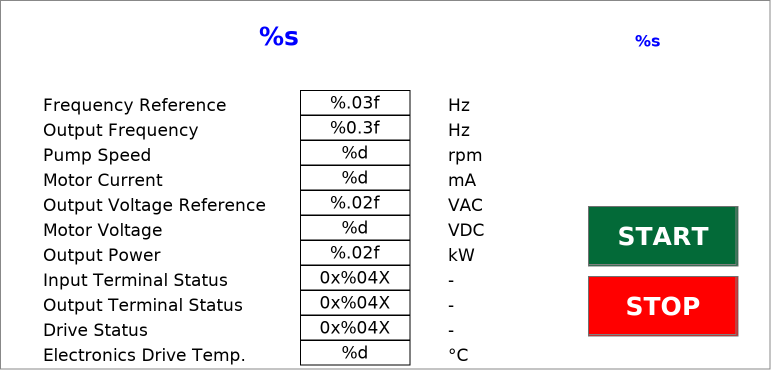
VISUALIZATION GUI_TEMPLATE_ECODRY_V01  // 771x370
VAR_IN_OUT
	m_Instance:	FB_CRYO_PUMP_ECODRY;
	m_bEnable:	BOOL;	// Flag to start/stop the pump
END_VAR
    Rectangle (300,90 110x25), "%.03f", text variable: m_Instance.stat.lrFreqRef
    Rectangle (300,115 110x25), "%0.3f", text variable: m_Instance.stat.lrOutFreq
    Rectangle (300,165 110x25), "%d", text variable: m_Instance.stat.nMotorCurr
    Rectangle (300,190 110x25), "%.02f", text variable: m_Instance.stat.lrOutVoltRef
    Label (40,90 245x30), "Frequency Reference"
    Label (40,115 245x30), "Output Frequency"
    Label (40,165 245x30), "Motor Current"
    Label (40,190 245x30), "Output Voltage Reference"
    Rectangle (300,215 110x25), "%d", text variable: m_Instance.stat.nMotorVolt
    Rectangle (300,240 110x25), "%.02f", text variable: m_Instance.stat.lrOutPower
    Rectangle (300,265 110x25), "0x%04X"
    Rectangle (300,290 110x25), "0x%04X"
    Label (40,215 245x30), "Motor Voltage"
    Label (40,240 245x30), "Output Power"
    Label (40,265 245x30), "Input Terminal Status"
    Label (40,290 245x30), "Output Terminal Status"
    Rectangle (300,315 110x25), "0x%04X"
    Rectangle (300,340 110x25), "%d", text variable: m_Instance.stat.nElecTemp
    Label (40,315 245x30), "Drive Status"
    Label (40,340 245x30), "Electronics Drive Temp."
    Label (445,90 59x30), "Hz"
    Label (445,115 59x30), "Hz"
    Label (445,165 59x30), "mA"
    Label (445,190 59x30), "VAC"
    Label (445,215 59x30), "VDC"
    Label (445,240 59x30), "kW"
    Label (445,265 59x30), "-"
    Label (445,290 59x30), "-"
    Label (445,315 59x30), "-"
    Label (445,340 59x30), "°C"
    Rectangle (164,21 230x30), "%s", text variable: m_Instance.in_sName
    Button (588,206 150x60), "START"
        OnMouseClick: execute { m_bEnable := TRUE; }
    Button (588,276 150x60), "STOP"
        OnMouseClick: execute { m_bEnable := FALSE; }
    Rectangle (525,26 246x30), "%s", tooltip "Control Mode", text variable: m_Instance.stat.sPumpState
    Rectangle (300,140 110x25), "%d", text variable: m_Instance.stat.nPumpSpeed
    Label (40,140 245x30), "Pump Speed"
    Label (445,140 59x30), "rpm"
END_VISUALIZATION

(* stored: Version 1.1.0.1, ProductVersion 3.1.4024.9
   Visu GUI_TEMPLATE_ECODRY_V01: Id {f8b19496-61df-474f-a9f9-5512734b92f0} *)
